TYPE ref_sv_input :
STRUCT
	in_flg_sensA:	BOOL;
	in_flg_sensB:	BOOL;
END_STRUCT
END_TYPE

(* stored: Version 1.1.0.1, ProductVersion 3.1.4024.11
   DUT ref_sv_input: Id {8eab64bc-78ef-43a0-b6ae-1d3d1aaddb5d} *)
